// TIA Portal V20 export
FUNCTION_BLOCK "LER_PowerMeter_7KM"   // FB175, LAD
// stored: Access Published, MemoryReserve 100, SetENOAutomatically false
   VAR_INPUT
      unitMode : DInt;   // Requested unit mode
   END_VAR
   VAR_OUTPUT
      Error : Bool;
      status : Word;
   END_VAR
   VAR_IN_OUT
      configuration : "LER_typePAC3220Configuration";
      controlNode : "LER_typePAC3220ControlNode";
      moduleInterface : "LER_typePAC3220Interface";
   END_VAR
   VAR
      statInput_Status : "LER_typePAC3220Input_Status";
      statOuput_Status : "LER_typePAC3220Output_Status";
      statRetValWord { S7_SetPoint := 'True'} : Array[1..#count] of Word;
      statRetValInt : Array[1..#count] of Int;
   END_VAR
   VAR_TEMP
      tempRET_VAL : Array[1..#count] of Word;
      tempIndex : Int;
   END_VAR
   VAR CONSTANT
      count : Int := 2;
      True : Bool := true;   // OEM: replace with ProDiag statuses that command unit state
      False : Bool;   // OEM: replace with ProDiag statuses that command unit state
      STATUS_NO_ERROR_OCCURRED : Word;   // No error occurred.
      ERR_HWID_NOT_CONFIGURED : Word := 16#8090;   // You have not configured a module for the specified hardware identifier or You have ignored the restriction concerning the length of consistent data, or you have not specified a hardware identifier as an address at parameter LADDR
      ERR_RECORD_DATA_TYPE : Word := 16#8092;   // Non-supported data type in the RECORD parameter.
      ERR_NO_DP_PROFINET_IO_MOUDLE : Word := 16#8093;   // No DP module/PROFINET IO device from which you can read consistent data exists for the hardware identifier specified in LADDR . This error code also occurs if the module addressed by means of LADDR does not have inputs.
      ERR_IO_ACCESS_PERMISSION : Word := 16#80A0;   // An access error was detected when accessing the I/O.
      ERR_ERCORD_LENGTH_INSUFFICIENT : Word := 16#80B1;   // The length of the specified destination area at parameter RECORD is shorter than the configured user data length.
      ERR_DATA_NOT_RECEIVED : Word := 16#80C0;   // The data have not been read yet.
   END_VAR
BEGIN

REGION Network 1 (SCL): ###### Hardwere ID mapping #######
   #statRetValInt[1] := DPRD_DAT(LADDR := #configuration."Basic type 3_HW_ID", RECORD => #statInput_Status);
   #statRetValInt[2] := DPRD_DAT(LADDR := #configuration."Basic type 3_HW_ID", RECORD => #statOuput_Status);
END_REGION

REGION Network 2 (SCL): Error Check
   REGION  Error Code Search

       // Hardwere ID mapping Error
       IF (#statRetValWord <> #tempRET_VAL) THEN
           FOR #tempIndex := 1 TO #count DO
               CASE #statRetValWord[#tempIndex] OF

               #ERR_HWID_NOT_CONFIGURED:
               #status := #ERR_HWID_NOT_CONFIGURED;

               #ERR_RECORD_DATA_TYPE:
               #status := #ERR_RECORD_DATA_TYPE;

               #ERR_NO_DP_PROFINET_IO_MOUDLE:
               #status := #ERR_NO_DP_PROFINET_IO_MOUDLE;

               #ERR_IO_ACCESS_PERMISSION:
               #status := #ERR_IO_ACCESS_PERMISSION;

               #ERR_ERCORD_LENGTH_INSUFFICIENT:
               #status := #ERR_ERCORD_LENGTH_INSUFFICIENT;

               #ERR_DATA_NOT_RECEIVED:
               #status := #ERR_DATA_NOT_RECEIVED;

               END_CASE;
               EXIT;
           END_FOR;

       ELSE
           #status := #STATUS_NO_ERROR_OCCURRED;

       END_IF;

   END_REGION


   // Error Bit
   #Error := #status <> 0;
END_REGION

REGION Network 3 (SCL): ##### Outputs mapping #####
   // moduleInterface, controlNode Data Move
   #moduleInterface.monitoring.Input_Status := #controlNode.monitoring.Input_Status := #statInput_Status;
   #moduleInterface.monitoring.Ouput_Status := #controlNode.monitoring.Ouput_Status := #statOuput_Status;
   #moduleInterface.monitoring.Error := #controlNode.monitoring.Error := #Error;
END_REGION
END_FUNCTION_BLOCK
